{attribute 'linkalways'} 
{attribute 'no_explicit_call' := 'This FB is a CLASS and must be accessed using methods or properties'}
{attribute 'enable_dynamic_creation'}
FUNCTION_BLOCK FINAL ABS_LINT EXTENDS Node
VAR
	in : _LINT(0);
	out : _LINT(0);
END_VAR

METHOD PUBLIC Clone : I_Node
VAR
	pNode : POINTER TO ABS_LINT;
END_VAR
pNode := __NEW(ABS_LINT);
Clone := pNode^;
END_METHOD

METHOD FB_init : BOOL
VAR_INPUT
	bInitRetains : BOOL; // if TRUE, the retain variables are initialized (warm start / cold start)
	bInCopyCode : BOOL;  // if TRUE, the instance afterwards gets moved into the copy code (online change)
END_VAR
AddInput('in',THIS^.in);
AddOutput('out', THIS^.out);
END_METHOD

METHOD PROTECTED OnExecute
VAR
END_VAR
out.Value := ABS(in.Value);
END_METHOD

END_FUNCTION_BLOCK

(* stored: Version 1.1.0.1, ProductVersion 3.1.4024.15
   POU ABS_LINT: Id {4f4bfeba-ffef-4285-866e-a38e6b79c097}, SpecialFunc None
   Folder Constructor: Id {a39add6d-5cd0-436a-ace3-bc09535bbf6b}
   Method Clone: Id {caf8c478-1d4a-4cb2-8c8e-2a10597a503b}
   Method FB_init: Id {10004088-064e-4dd0-a129-ebfbf0e6e2c1}
   Method OnExecute: Id {895e9fb7-d4a5-4bb3-b2b9-c261e7f5f8f7} *)
